// TIA Portal V20 export
DATA_BLOCK "EeMonitorData"   // DB108
TITLE = EeMonitorData
AUTHOR : SICAR
FAMILY : DB
// Energy efficency monitor Daten / Energy efficency monitor data
// stored: InstanceOfName LSicar_typeEemData, InstanceOfType UDT
"LSicar_typeEemData"
   // VAR
   //    machineConfiguration : EnS_EEm_typeConfig;
   //    machineOperation : EnS_EEm_typeOperation;
   //    measConfiguration : Array[0..9] of EnS_EEm_typeMeasConfig;
   //    measOperation : Array[0..9] of EnS_EEm_typeMeasOperation;
   //    internalData : "LSicar_typeEemDataInternal";
   //    calcError : Bool;
   //    calcStatus : Word;
   //    calcRetVal : Int;
   //    reportCreateCsv : Bool;
   //    reportStatus : Word;
   //    reportNameCsv : String[80];
   // END_VAR
BEGIN
   machineConfiguration.eStateName[1] := 'Auto';
   machineConfiguration.eStateName[2] := 'Auto Preselect';
   machineConfiguration.eStateName[3] := 'Manual';
   machineConfiguration.eStateName[4] := 'Idle';
   machineConfiguration.eStateName[5] := 'Fault';
   machineConfiguration.eStateName[6..7] := '-Not used-';
   machineOperation.maskEnPI := 16#0002;
   measConfiguration[2]."name" := 'PAC Electrical Infeed';
   measConfiguration[3..9]."name" := 'MeasPointXX';
   measConfiguration[2].nameShort := 'P01';
   measConfiguration[3..9].nameShort := 'XX01';
   measConfiguration[2..9].media := 'electrical';
   measConfiguration[2..9].unitCounterNumber := 1;
   measConfiguration[2..9].unitCounterText := 'Wh';
   measConfiguration[2..9].unitActValueNumber := 0;
   measConfiguration[2..9].unitActValueText := 'W';
   measConfiguration[2..9].inputType := 1;
   measConfiguration[2..9].type1Counter.overflowCntValue := 1000000.0;
   measConfiguration[2..9].type1Counter.normFactor := 1.0;
   internalData.productiveEnergyStates[1] := true;
END_DATA_BLOCK
